{attribute 'qualified_only'}
VAR_GLOBAL
	bTaskRunning : BOOL;
END_VAR

(* stored: Version 1.1.0.1, ProductVersion 3.1.4024.12
   GVL GVL_SIMU: Id {61b9c5e6-84eb-4749-93b4-c4a868ecb108} *)
